TEXTLIST AxesDialogRotUnitsTextList
  0 = 'd / m / s'
  1 = 'degrees'
  2 = 'radians'
   = ''
END_TEXTLIST

(* stored: Version 1.1.0.1, ProductVersion 3.1.4019.2
   TextList AxesDialogRotUnitsTextList: Id {fbf7886e-c2e5-4c62-b715-4cb45f7ead93} *)
